// TwinCAT 3 PLC project PLC_01
// ProgramVersion: 3.1.4020.4
// libraries:
//   Tc2_Standard, * (Beckhoff Automation GmbH)
//   Tc2_System, * (Beckhoff Automation GmbH)
//   Tc2_Utilities, * (Beckhoff Automation GmbH)
//   Tc3_Module, * (Beckhoff Automation GmbH)
//   VisuDialogs, * (System)
// project tree:
//   DUTs/System/ ST_Ctrl.TcDUT, ST_Error.TcDUT, ST_Status.TcDUT
//   / GlobalTextList.TcGTLO, PlcTask.TcTTO, Visualisierungsmanager.TcVMO (not stored), VISU_TASK.TcTTO
//   GVLs/ GVL_Const.TcGVL
//   POUs/700 File/ FB_DirectoryRead.TcPOU, FB_openPDF.TcPOU
//   POUs/800 Visualisierung/ FB_TrendBuffer.TcPOU, PRG_System.TcPOU, PRG_Visualisierung.TcPOU
//   POUs/ FB_PWM.TcPOU, FUN_String_to_Time.TcPOU, MAIN.TcPOU, PRG_CAN.TcPOU
//   VISUs/ Frame_Trend_Einzel.TcVIS, Visualization.TcVIS
// real-time tasks:
//   TASK PlcTask: cycle T#10ms, priority 20, ADS port 350
//   TASK VISU_TASK: cycle T#200000us, priority 30, ADS port 351
// I/O:
//   DEVICE Gerät 1 (EtherCAT), AmsNetId 5.42.100.143.2.1
//     Klemme 1 (EK1200) [EK1200-5000 EtherCAT Netzteil (2A E-Bus)]
//       Klemme 2 (EL2008) [EL2008 8K. Dig. Ausgang 24V, 0.5A]
//       Klemme 3 (EL2008) [EL2008 8K. Dig. Ausgang 24V, 0.5A]
//       Klemme 4 (EL4104) [EL4104 4Ch. Ana. Ausgang 0-10V, 16bit]
//       Klemme 5 (EL3162) [EL3162 2K. Ana. Eingang 0-10V]
//       Klemme 6 (EL6751) [EL6751 (CANopen Master)]
//       Klemme 7 (EL9011) [EL9011 Endklemme]
//   DEVICE Gerät 2 (EL6751), AmsNetId 5.42.100.143.3.1
//     Box 8 (CANopen Node)
// variable links:
//   PLC_01/PLC_01 Instance <-> Device 1 (EtherCAT)/Term 1 (EK1200)/Term 2 (EL2008)
//     PlcTask Outputs/MAIN.ATQ_output1 <-> Channel 1/Output
//     PlcTask Outputs/MAIN.ATQ_output2 <-> Channel 2/Output
//   PLC_01/PLC_01 Instance <-> Device 1 (EtherCAT)/Term 1 (EK1200)/Term 6 (EL6751)
//     PlcTask Inputs/MAIN.ATI_input1 <-> WcState/WcState
//   PLC_01/PLC_01 Instance <-> Device 2 (EL6751)/Box 8 (CANopen Node)
//     PlcTask Inputs/PRG_CAN.CAN_master_Rx_ATI_1040 <-> TxPDO 1/Inputs/#10.40
//     PlcTask Inputs/PRG_CAN.CAN_master_Rx_ATI_201 <-> TxPDO 1/Inputs/#2.01
//     PlcTask Outputs/PRG_CAN.CAN_master_Tx_ATQ_121 <-> RxPDO 1/Outputs/#1.21
//     PlcTask Outputs/PRG_CAN.CAN_master_Tx_ATQ_642 <-> RxPDO 1/Outputs/#6.42

CONFIGURATION PLC_01
    RESOURCE PLC ON TwinCAT3
        TASK PlcTask(INTERVAL := T#10ms, PRIORITY := 20);
        TASK VISU_TASK(INTERVAL := T#200000us, PRIORITY := 30);
        PROGRAM MAIN WITH PlcTask : MAIN;
        PROGRAM VisuElems_Visu_Prg WITH VISU_TASK : VisuElems.Visu_Prg;
    END_RESOURCE
END_CONFIGURATION

// ---- DUTs/System/ST_Ctrl.TcDUT
TYPE ST_Ctrl :
STRUCT
	Init: BOOL;
	Execute: BOOL;
	Reset: BOOL;
	

END_STRUCT
END_TYPE

// ---- DUTs/System/ST_Error.TcDUT
TYPE ST_Error :
STRUCT
	Err				: BOOL;			// Hier wird das Auftreten eines Fehlers signalisiert
	ID				: UDINT;		// Hier wird eine codierte Fehlermeldung bereitgestellt - mehrere Fehler gleichzeitig möglich
	Ort				: STRING;		// Bei gesetztem Error die Angabe Ort
	OrtID			: UDINT;		// Bei gesetztem Error die Angabe Ort Id
	Modul			: STRING;		// Bei gesetztem Error die Angabe Modul
	ModulID			: UDINT;		// Bei gesetztem Error die Angabe Modul Id
	SubModul		: STRING;		// Bei gesetztem Error die Angabe SubModul
	SubModulID		: UDINT;		// Bei gesetztem Error die Angabe SubModul Id
	Text			: STRING;		// Hier wird die erste Fehlermeldung als Text bereitgestellt - nur eine Meldung möglich
	TextID			: UDINT;		// Hier wird die erste Fehlermeldung als Text bereitgestellt - nur eine Meldung möglich
	SystemTime		: STRING;		// Bei gesetztem Error die Angabe der Zeit = Systemzeit, String = YYYY-MM-DD-hh:mm:ss:xxx
													

END_STRUCT
END_TYPE

// ---- DUTs/System/ST_Status.TcDUT
TYPE ST_Status :
STRUCT
	InitOk:BOOL;
	Done:BOOL;
	Busy:BOOL;
	stError:ST_Error;

END_STRUCT
END_TYPE

// ---- GVLs/GVL_Const.TcGVL
VAR_GLOBAL CONSTANT
	
//Trend Darstellung
	gc_max_Plots				: INT:=2; 	//Maximale Anzahl an FB Trend Instanzen (und somit an möglichen Plots)
	gc_Max_ITEMS				: INT:=500; //Maximale Anzahl an Items (bei 50 wird nur das halbe Histogramm gefüllt)

//Directory read
	gcFileList_Min		: UINT:=1;						(*First line of the table*)
	gcFileList_Max		: UINT:=100;					(*Last line of the table*)
END_VAR

// ---- POUs/MAIN.TcPOU
PROGRAM MAIN
VAR

	
	//Digital I/O
	ATI_input1 AT%I* : BOOL;
	ATI_input2 AT%I* : BOOL;
	
	ATQ_output1 AT%Q* : BOOL;
	ATQ_output2 AT%Q* : BOOL;
	
	

	
	
	
	
	//zu öffnende Datei
	dateiname:STRING:='C:\Temp\B.pdf';		//Variante 1
	dateiname2:STRING:='';									//Variante 2 (wird aus Pfad und gefundener Datei zusammengesetzt
	Pfadname: STRING:='C:\Temp\';							//zu durchsuchender Pfad
	dateiindex:UINT;										//index der zu wählenden Datei
	
	//PWM Zeiten
	szeit_on:STRING:='500';		//als String (Eingabe in Visu)
	tzeit_on:TIME;				//als Zeit (umgerechnet mit der Funktion String_to_Time)
	szeit_off:STRING:='500';
	tzeit_off:TIME;
	
	// Auswahlbox
	auswahl_index: INT;			//gewählter index
	auswahl : ARRAY[0..2] OF STRING:=['Ein', 'Aus', 'PWM'];	//zur Auswahl stehende Betriebsarten
	
	//Instanzen:
	fbpwm: FB_PWM;
	
	fbdirectoryRead		: FB_DirectoryRead;
	fbopenPDF		 	: FB_openPDF;
	fbopenPDF2			: FB_openPDF;
	
	
	ctrl_pdf_1: ST_Ctrl;
	ctrl_pdf_2: ST_Ctrl;
	ctrl_readdir: ST_Ctrl;
	status:ST_Status;
	
	
	step: INT;
	change: BOOL;
	step_last: INT;
	
	plot : ARRAY[1..GVL_Const.gc_max_Plots] OF REAL;
	
	
END_VAR


PRG_System();

//Aufruf des Programms zum öffnen der PDF Datei (direkte Pfadangabe)
fbopenPDF(
	ctrl:=ctrl_pdf_1,				//ctrl.Execute startet den Öffnen Vorgang
	dateiname:=dateiname,	//Pfad zu der zu öffnenden Datei
	status=>status );		//Rückgabe des Status

//Über Verzeichnis auslesen
fbdirectoryRead(ctrl:=ctrl_readdir , PathName:=Pfadname , status=> );
//Dateiauswählen
dateiname2:=Tc2_Standard.CONCAT(Pfadname,fbdirectoryRead.List[dateiindex]);
//und öffnen
fbopenPDF2(
	ctrl:=ctrl_pdf_2,		//ctrl.Execute startet den Öffnen Vorgang
	dateiname:=dateiname2,	//Pfad zu der zu öffnenden Datei
	status=>status );		//Rückgabe des Status

//Aufruf des Plot Diagramms	
plot[1]:=BOOL_TO_REAL(ATQ_output1);
plot[2]:=BOOL_TO_REAL(ATQ_output2);
PRG_Visualisierung(plot:=plot , TaskCycleTime_ms:=PRG_System.TaskCycleTime_ms );	

//Betriebsartenauswahl
CASE step OF
	100: //idle
		IF auswahl_index<>step_last THEN
			CASE auswahl_index OF
			0:	step:=0;
				step_last:=0;
			1: 	step:=1;
				step_last:=1;
			2:  step:=2;
				step_last:=2;
			END_CASE
		END_IF
		
	0: //Ein
		ATQ_output1:=TRUE;
		ATQ_output2:=TRUE;
		step:=100;
		
	1: // Aus
		ATQ_output1:=FALSE;
		ATQ_output2:=FALSE;
		step:=100;
		
	2: //PWM	
		//UMrechnung der String in Zeiten
		tzeit_on:=FUN_String_to_Time(text:=szeit_on);
		tzeit_off:=FUN_String_to_Time(text:=szeit_off);
		
		fbpwm(
			tHightime:=tzeit_on,	//High Zeit
			tLowtime:=tzeit_off);	//Low Zeit
		ATQ_output2:=fbpwm.output;	//Schreiben des Ausgangs
		
		IF auswahl_index<>2 THEN
			step:=100;
		END_IF
END_CASE


PRG_CAN();

END_PROGRAM

// ---- POUs/FB_PWM.TcPOU
FUNCTION_BLOCK FB_PWM
VAR_INPUT
	tHightime	: TIME;
	tLowtime	: TIME;

END_VAR
VAR_OUTPUT
	output		: BOOL;
END_VAR
VAR
 	timer 		: Tc2_Standard.TON;
	step		: INT;
END_VAR


CASE step OF
	0:	//low
		output:=FALSE;
		timer(IN:=TRUE , PT:=tLowtime , Q=> , ET=> );
		IF timer.Q THEN
			timer(IN:=FALSE);
			step:=1;
		END_IF
		
	1: 	//high
		output:=True;
		timer(IN:=TRUE , PT:=tHightime , Q=> , ET=> );
		IF timer.Q THEN
			timer(IN:=FALSE);
			step:=0;
		END_IF
END_CASE

END_FUNCTION_BLOCK

// ---- POUs/700 File/FB_DirectoryRead.TcPOU
FUNCTION_BLOCK FB_DirectoryRead
VAR_INPUT
	ctrl: ST_Ctrl;
	PathName : STRING;
END_VAR
VAR_OUTPUT
	status		: ST_Status;
	List		: ARRAY[gcFileList_Min..gcFileList_Max] OF STRING;
END_VAR
VAR
	nstep: INT;
	
	fbEnumFindFileList			: FB_EnumFindFileList;
	sPathName: STRING(255);
	FindList 						: ARRAY[gcFileList_Min..gcFileList_Max] OF ST_FindFileEntry;
	nindex: UINT;
END_VAR

CASE nstep OF
0: //init
	status.InitOk:=TRUE;
	
	IF status.InitOk THEN
		nstep:=1;
	END_IF
	
1: //idle
	
	IF ctrl.Execute THEN
		status.Done:=FALSE;
		status.Busy:=TRUE;
		nstep:=2;
	END_IF
	
2: //lesen öffnen
	sPathName:=CONCAT(PathName, '*.pdf') ;	

	fbEnumFindFileList(
		sNetId:='',
		sPathName:=sPathName ,
		eCmd:=eEnumCmd_First ,
		pFindList:=ADR(FindList) ,
		cbFindList:=SIZEOF(FindList) ,
		bExecute:=TRUE ,
		tTimeout:= ,
		bBusy=> ,
		bError=> ,
		nErrID=> ,
		bEOE=>  ,
		nFindFiles=> );

	// Abfrage ob Fertig und kein Fehler
	IF NOT fbEnumFindFileList.bBUSY THEN
		status.Busy:=FALSE;
		IF NOT fbEnumFindFileList.bError THEN
			fbEnumFindFileList(bExecute:=FALSE);
			IF fbEnumFindFileList.bEOE THEN
				
				FOR nindex:=gcFileList_Min TO gcFileList_Max DO
					List[nindex]:=FindList[nindex].sFileName;
				END_FOR
				
				nstep:=3;
			END_IF
		ELSE
			nstep:=99; //Fehler
		END_IF
		
	END_IF	
	
	
3: //fertig
	status.Busy:=FALSE;
	status.Done:=TRUE;
	IF NOT ctrl.Execute THEN
		nstep:=1;
	END_IF

8: //reset
	status.stError.Err:=FALSE;
	fbEnumFindFileList(bExecute:=FALSE);
	nstep:=0;

99: //Fehler
	status.stError.Err:=TRUE;
	status.stError.ID:=fbEnumFindFileList.nErrID;
	status.Busy:=FALSE;
	
	IF ctrl.Reset THEN
		nstep:=8;
	END_IF
	
END_CASE

END_FUNCTION_BLOCK

// ---- POUs/700 File/FB_openPDF.TcPOU
FUNCTION_BLOCK FB_openPDF
VAR_INPUT
	ctrl: ST_Ctrl;
	dateiname:STRING:='C:\Temp\Beispielprojekt.pdf';
END_VAR

VAR_OUTPUT
	status: ST_Status;
END_VAR

VAR
	fbntstartprozess: NT_StartProcess;
	nstep: INT;
END_VAR

CASE nstep OF
0: //init
	status.InitOk:=TRUE;
	
	IF status.InitOk THEN
		nstep:=1;
	END_IF
	
1: //idle
	
	IF ctrl.Execute THEN
		status.Done:=FALSE;
		status.Busy:=TRUE;
		nstep:=2;
	END_IF
	
2: //PDF öffnen
	
	fbntstartprozess(
		NETID:='' , 
		(*64 Bit*)
		//PATHSTR:='C:\Program Files (x86)\Adobe\Acrobat Reader DC\Reader\AcroRd32.exe' , //Pfad des PDF Viewers
		//DIRNAME:='C:\Program Files (x86)\' , 											//Verzeichnis des Viewers
		(**)
		(*32 Bit*)
		PATHSTR:='C:\Program Files\Adobe\Acrobat Reader DC\Reader\AcroRd32.exe' , //Pfad des PDF Viewers
		DIRNAME:='C:\Program Files\' , 											//Verzeichnis des Viewers
		(**)
		COMNDLINE:=dateiname ,  												//zu öffnende Datei
		START:= TRUE, 
		TMOUT:= , 																//Default wert
		BUSY=> , 
		ERR=> , 
		ERRID=> );

	// Abfrage ob Fertig und kein Fehler
	IF NOT fbntstartprozess.BUSY THEN
		status.Busy:=FALSE;
		IF NOT fbntstartprozess.ERR THEN
			nstep:=3;
			fbntstartprozess(START:=FALSE);
		ELSE
			nstep:=99; //Fehler
		END_IF
		
	END_IF	
	
	
3: //fertig
	status.Busy:=FALSE;
	status.Done:=TRUE;
	IF NOT ctrl.Execute THEN
		nstep:=1;
	END_IF

8: //reset
	status.stError.Err:=FALSE;
	fbntstartprozess(START:=FALSE);
	nstep:=0;

99: //Fehler
	status.stError.Err:=TRUE;
	status.stError.ID:=fbntstartprozess.ERRID;
	status.Busy:=FALSE;
	
	IF ctrl.Reset THEN
		nstep:=8;
	END_IF
	
END_CASE

END_FUNCTION_BLOCK

// ---- POUs/800 Visualisierung/PRG_System.TcPOU
PROGRAM PRG_System
VAR_INPUT
	bWritePersistentData			: BOOL; //True, wenn persistente Daten geschrieben werden sollen
	bStartExplorer					: BOOL; //True, wenn Window Explorer geöffnet werden soll
	bShutdown						: BOOL; //True, wenn Rechner runtergefahren werden soll
END_VAR
VAR_OUTPUT
	SystemTime_ms					: STRING;
	TaskCycleTime_ms				: UDINT;
	SystemTime_DT					: DT;
	nCountPersistentData			: UINT;			//Zähler der persitenten Schreibvorgänge
	stError							: ST_Error;
END_VAR
VAR
	fbGetCurTaskIdx					: GETCURTASKINDEX;
	fbRegQueryValue					: FB_RegQueryValue;

	fbLocalSystemTime				: FB_LocalSystemTime;
	fbSetLocalTime 					: NT_SetLocalTime;
	fbGetTimeZoneInformation 		: FB_GetTimeZoneInformation;
	TaskCycleTime_ns				: UDINT;
	
	LastExecTime_ms					: UDINT;
	rtrigCycleTimeExceeded			: R_TRIG;
	
	
	rTrigPersistentDataWrite		: R_TRIG;
	fbWritePersistentData			: FB_WritePersistentData;
	rTrigPersistentDataDone			: F_TRIG;

	bFirstCycle						: BOOL;
	CountCycleTimeExceeded	: UINT;
	PeakHoldLastExectime_ms: UDINT;
	
	fbShutdown						: NT_Shutdown;
	fbStartProcess					: NT_StartProcess;
	
END_VAR

// ---------------------------------------------------------------------------------------------------------------------
// _AppInfo
// ---------------------------------------------------------------------------------------------------------------------
 (*
 TYPE PlcAppSystemInfo

	Each PLC provides a global instance of this type named '_AppInfo'.
	The corresponding namespace is 'TwinCAT_SystemInfoVarList'. For example this has to be added inside a library.

--------------------------------------------------------------------------------------------------------------------------------------------------------------------------------------------------------------------------------------------------
TYPE PlcAppSystemInfo
STRUCT
         ObjId             		: OTCID;				// 	object ID of the PLC project instance
         TaskCnt           		: UDINT;				// The number of tasks in the actual runtime system.
         OnlineChangeCnt   		: UDINT;				// The number of online changes made since the last complete download.
         Flags             		: DWORD;				// Reserved for future use
         AdsPort           		: UINT;					// ADS port of PLC application
         BootDataLoaded    		: BOOL;					// PERSISTENT variables: LOADED (without error)
         OldBootData       		: BOOL;					// PERSISTENT variables: INVALID (the back-up copy was loaded, since no valid data was present)
         AppTimestamp      		: DT;					// Date and time of application start
         KeepOutputsOnBP   		: BOOL;					// The flag can be set to avoid that the outputs are zero-filled if a breakpoint is reached. The task keeps running. Only the execution of PLC code is interrupted.
         TComSrvPtr        		: ITComObjectServer;	// Pointer to TcCOM Object Server
         AppName           		: STRING(63);			// TwinCAT generated name containing the port number
         ProjectName       		: STRING(63);			// The name of the PLC project.
END_STRUCT
END_TYPE
 
If the variable runTimeNo was used under TwinCAT 2, the program code has to be changed.
Sample:
Usage under TwinCAT 2:   nPlcAdsPort := 801 + (SystemInfo.runTimeNo - 1) * 10;
Usage under TwinCAT 3:   nPlcAdsPort := _AppInfo.AdsPort;
 *)
 
 _AppInfo.ObjId:=_AppInfo.ObjId;
 _AppInfo.TaskCnt:=_AppInfo.TaskCnt;
 _AppInfo.OnlineChangeCnt:=_AppInfo.OnlineChangeCnt;
 _AppInfo.Flags:=_AppInfo.Flags;
 _AppInfo.AdsPort:=_AppInfo.AdsPort;
 _AppInfo.BootDataLoaded:=_AppInfo.BootDataLoaded;
 _AppInfo.OldBootData:=_AppInfo.OldBootData;
 _AppInfo.AppTimestamp:=_AppInfo.AppTimestamp;
 _AppInfo.KeepOutputsOnBP:=_AppInfo.KeepOutputsOnBP;
 _AppInfo.TComSrvPtr:=_AppInfo.TComSrvPtr;
 _AppInfo.AppName:=_AppInfo.AppName;
 _AppInfo.ProjectName:=_AppInfo.ProjectName;


// ---------------------------------------------------------------------------------------------------------------------
// _TaskInfo
// ---------------------------------------------------------------------------------------------------------------------
 (*
 TYPE PlcTaskSystemInfo

	Each PLC provides an array of global instances of this type named '_TaskInfo[]'.
	The corresponding namespace is 'TwinCAT_SystemInfoVarList'. For example this has to be added inside a library.

--------------------------------------------------------------------------------------------------------------------------------------------------------------------------------------------------------------------------------------------------
{attribute 'Namespace' := 'PLC'}
TYPE PlcTaskSystemInfo
STRUCT
         ObjId             		: OTCID;				// 	Object ID of task reference calling the PLC program.
         CycleTime         		: UDINT;				// Cycletime set in the task configuration in parts of 100ns.
         Priority          		: UINT;					// Priority set in the task configuration.
         AdsPort           		: UINT;					// 	ADS port of Task
         CycleCount        		: UDINT;				// Cyclecounter.
         DcTaskTime        		: LINT;					// Distributed Clock System Time. It remains constant for a task duration.
         LastExecTime      		: UDINT;				// Needed cycletime for the last cycle in parts of 100ns.
         FirstCycle        		: BOOL;					// The variable is TRUE in the first cycle of the task.
         CycleTimeExceeded 		: BOOL;					// 	The variable is TRUE if the runtime of the task exceeds the cycletime set in task configuration.
         TaskName          		: STRING(63);			// Contains the name of the task
END_STRUCT
END_TYPE

Sample:
fbGetCurTaskIdx();                                                                           // declared as: fbGetCurTaskIdx : GETCURTASKINDEX;
nCycleTime := _TaskInfo[fbGetCurTaskIdx.index].CycleTime;
*)
 
 fbGetCurTaskIdx();                                                                           // declared as: fbGetCurTaskIdx : GETCURTASKINDEX;

 _TaskInfo[fbGetCurTaskIdx.index].ObjId:=_TaskInfo[fbGetCurTaskIdx.index].ObjId;
 _TaskInfo[fbGetCurTaskIdx.index].CycleTime:=_TaskInfo[fbGetCurTaskIdx.index].CycleTime;
 _TaskInfo[fbGetCurTaskIdx.index].Priority:=_TaskInfo[fbGetCurTaskIdx.index].Priority;
 _TaskInfo[fbGetCurTaskIdx.index].AdsPort:=_TaskInfo[fbGetCurTaskIdx.index].AdsPort;
 _TaskInfo[fbGetCurTaskIdx.index].CycleCount:=_TaskInfo[fbGetCurTaskIdx.index].CycleCount;
 _TaskInfo[fbGetCurTaskIdx.index].DcTaskTime:=_TaskInfo[fbGetCurTaskIdx.index].DcTaskTime;
 _TaskInfo[fbGetCurTaskIdx.index].LastExecTime:=_TaskInfo[fbGetCurTaskIdx.index].LastExecTime;
 _TaskInfo[fbGetCurTaskIdx.index].FirstCycle:=_TaskInfo[fbGetCurTaskIdx.index].FirstCycle;
 _TaskInfo[fbGetCurTaskIdx.index].CycleTimeExceeded:=_TaskInfo[fbGetCurTaskIdx.index].CycleTimeExceeded;
 _TaskInfo[fbGetCurTaskIdx.index].TaskName:=_TaskInfo[fbGetCurTaskIdx.index].TaskName;
 
// ---------------------------------------------------------------------------------------------------------------------
// Zykluszeit mit Spitzenwert 8Peak Hold)
// ---------------------------------------------------------------------------------------------------------------------
TaskCycleTime_ns:=_TaskInfo[fbGetCurTaskIdx.index].CycleTime/10;
TaskCycleTime_ms:=_TaskInfo[fbGetCurTaskIdx.index].CycleTime/10000;
LastExecTime_ms:=_TaskInfo[fbGetCurTaskIdx.index].LastExecTime/10000;
IF PeakHoldLastExectime_ms<LastExecTime_ms THEN
	PeakHoldLastExectime_ms:=LastExecTime_ms;
END_IF

// ---------------------------------------------------------------------------------------------------------------------
// Zykluszeitüberschreitungen zählen
// ---------------------------------------------------------------------------------------------------------------------
rtrigCycleTimeExceeded(CLK:=_TaskInfo[fbGetCurTaskIdx.index].CycleTimeExceeded , Q=> );
IF rtrigCycleTimeExceeded.Q THEN
	CountCycleTimeExceeded:=CountCycleTimeExceeded+1;
END_IF

// ---------------------------------------------------------------------------------------------------------------------
// PLC First Cycle
// ---------------------------------------------------------------------------------------------------------------------
bFirstCycle:=_TaskInfo[fbGetCurTaskIdx.index].FirstCycle;

// ---------------------------------------------------------------------------------------------------------------------
// Windows Systemzeit 
// ---------------------------------------------------------------------------------------------------------------------
 fbLocalSystemTime(
	sNetID:='' ,
	bEnable:=TRUE ,
	dwCycle:= ,
	dwOpt:= ,
	tTimeout:=DEFAULT_ADS_TIMEOUT ,
	bValid=> ,
	systemTime=> ,
	tzID=> );
IF fbLocalSystemTime.bValid THEN
	SystemTime_ms:=LEFT(SYSTEMTIME_TO_STRING(fbLocalSystemTime.systemTime),16);
	SystemTime_DT:=SYSTEMTIME_TO_DT(fbLocalSystemTime.systemTime);
END_IF

// ---------------------------------------------------------------------------------------------------------------------
// Persisten Data
// ---------------------------------------------------------------------------------------------------------------------
rTrigPersistentDataWrite(CLK:=bWritePersistentData , Q=> );
fbWritePersistentData(
	NETID:= '', 
	PORT:= _TaskInfo[fbGetCurTaskIdx.index].AdsPort , 
	START:= rTrigPersistentDataWrite.Q , 
	TMOUT:= DEFAULT_ADS_TIMEOUT , 
	MODE:= SPDM_2PASS, 
	BUSY=> , 
	ERR=> , 
	ERRID=> );
rTrigPersistentDataDone(CLK:=fbWritePersistentData.BUSY , Q=> );
IF rTrigPersistentDataDone.Q THEN
	nCountPersistentData:=nCountPersistentData+1;
END_IF

// ---------------------------------------------------------------------------------------------------------------------
// Windows / Explorer
// ---------------------------------------------------------------------------------------------------------------------
fbStartProcess(
	NETID:='' , 
	PATHSTR:='C:\Windows\Explorer.exe' , 
	DIRNAME:= , 
	COMNDLINE:= , 
	START:=bStartExplorer , 
	TMOUT:=DEFAULT_ADS_TIMEOUT , 
	BUSY=> , 
	ERR=> , 
	ERRID=> );





// ---------------------------------------------------------------------------------------------------------------------
// Windows / PC ausschalten
// ---------------------------------------------------------------------------------------------------------------------
fbShutdown(
	NETID:='' , 
	DELAY:=5 , 
	START:=bShutdown , 
	TMOUT:=DEFAULT_ADS_TIMEOUT , 
	BUSY=> , 
	ERR=> , 
	ERRID=> );


// ---------------------------------------------------------------------------------------------------------------------
// ENDE
// ---------------------------------------------------------------------------------------------------------------------

METHOD GetSystemTime : DT
VAR_INPUT
END_VAR
GetSystemTime:=SystemTime_DT;
END_METHOD

END_PROGRAM

// ---- POUs/800 Visualisierung/PRG_Visualisierung.TcPOU
PROGRAM PRG_Visualisierung
VAR_INPUT
	plot : ARRAY[1..GVL_Const.gc_max_Plots] OF REAL; 	//Array von den Werten (in REAL) die geplottet werden sollen
	TaskCycleTime_ms : UDINT;							//Zykluszeit in ms ( z.B. aus PRG_System)
END_VAR
VAR_OUTPUT
END_VAR
VAR
	
	fbpwmTrend :ARRAY[1..GVL_Const.gc_max_Plots] OF  FB_TrendBuffer;
	
	nindex:INT;
	
END_VAR


//Aufruf des FB zur Erzeugung des Trends
FOR nindex:=1  TO GVL_Const.gc_max_Plots DO  
	
	fbpwmTrend[nindex](
		uiValue:= plot[nindex],  						// Eingangssignal
		dtSystemTime:= PRG_System.GetSystemTime(), 
		tCycleTime:= UDINT_TO_TIME(TaskCycleTime_ms), 	// Zykluszeit
		bReverseFilll:= , 
		count=> , 
		dtFirstTimeStamp=> , 
		dtLastTimeStamp=> 
	);
END_FOR

END_PROGRAM

// ---- POUs/800 Visualisierung/FB_TrendBuffer.TcPOU
FUNCTION_BLOCK FB_TrendBuffer
VAR_INPUT
	uiValue 		: REAL;			//Zu plottender Wert
	dtSystemTime 	: DT;
	tCycleTime 		: TIME;			//Zyklus Zeit
	bReverseFilll 	: BOOL;			//False: von rechts nach links , True von Links nach rechts verschieben
END_VAR
VAR_OUTPUT
	count 		     : UINT;
	dtFirstTimeStamp : DT;
	dtLastTimeStamp  : DT;
END_VAR

VAR
	itemValue 		 : ARRAY[1..GVL_Const.gc_Max_ITEMS] OF REAL; 		//Array was an das Histogramm weitergegeben werden muss
	itemTimeStamp    : ARRAY[1..GVL_Const.gc_Max_ITEMS] OF DT;

	cycle 			 : TOF;
	bFullBuffer 	 : BOOL;
END_VAR

(*
- Pro zu Plottendem Wert ist eine Instanz anzulegen
- uiValue ist die Eingangsvariable
- itemValue ist das zu plottende Array

*)



IF NOT cycle.Q THEN
	count := MIN(count +1,GVL_Const.gc_Max_ITEMS);
	CASE BOOL_TO_INT(bReverseFilll) OF
	0:
		IF bFullBuffer THEN
			MEMCPY(ADR(itemValue),ADR(itemValue)+SIZEOF(itemValue[GVL_Const.gc_Max_ITEMS]),SIZEOF(itemValue)-SIZEOF(itemValue[GVL_Const.gc_Max_ITEMS]));
			MEMCPY(ADR(itemTimeStamp),ADR(itemTimeStamp)+SIZEOF(itemTimeStamp[GVL_Const.gc_Max_ITEMS]),SIZEOF(itemTimeStamp)-SIZEOF(itemTimeStamp[GVL_Const.gc_Max_ITEMS]));
		END_IF
		bFullBuffer := (count >= GVL_Const.gc_Max_ITEMS);
		itemValue[count] := uiValue;
		itemTimeStamp[count] := dtSystemTime;
	ELSE
		MEMCPY(ADR(itemValue)+SIZEOF(itemValue[GVL_Const.gc_Max_ITEMS]),ADR(itemValue),SIZEOF(itemValue)-SIZEOF(itemValue[GVL_Const.gc_Max_ITEMS]));
		MEMCPY(ADR(itemTimeStamp)+SIZEOF(itemTimeStamp[GVL_Const.gc_Max_ITEMS]),ADR(itemTimeStamp),SIZEOF(itemTimeStamp)-SIZEOF(itemTimeStamp[GVL_Const.gc_Max_ITEMS]));
		itemValue[1] := uiValue;
		itemTimeStamp[1] := dtSystemTime;
	END_CASE
	
	dtFirstTimeStamp := itemTimeStamp[1];
	dtLastTimeStamp := itemTimeStamp[count];
END_IF

cycle(IN:=NOT cycle.Q, PT:=tCycleTime);

END_FUNCTION_BLOCK

// ---- POUs/FUN_String_to_Time.TcPOU
FUNCTION FUN_String_to_Time : Time
VAR_INPUT
	text:STRING;
END_VAR
VAR
	temp :string;
END_VAR

//zusammensetzten des Strings
temp:=Tc2_Standard.CONCAT(STR1:=Tc2_Standard.CONCAT(STR1:='T#',STR2:=text),STR2:='ms');

//Konvertierung in Zeit
FUN_String_to_Time:=STRING_TO_TIME(temp);

END_FUNCTION

// ---- POUs/PRG_CAN.TcPOU
PROGRAM PRG_CAN
VAR_INPUT

END_VAR

VAR_OUTPUT

END_VAR

VAR
//CAN test
	//wird vom Master empfangen
	CAN_master_Rx_ATI_1040 	AT%I* :DINT;	// status word
	CAN_master_Rx_ATI_201   AT%I* :DINT;	// post-ramp speed	
	
	//wird vom Master gesendet
	CAN_master_Tx_ATQ_642 	AT%Q* :DINT;	// control word
	CAN_master_Tx_ATQ_121 	AT%Q* :DINT;	// digital speed	
	

(*
	Polled channel 			Data word 	Mapping parameter 	Size(bits) 		Default mapping status
	IN  channel 0 RxPDO 	Word 0, 1 	Pr MM.10 			32 				1040 (Pr 10.40, status word)
	IN  channel 1 RxPDO 	Word 2, 3 	Pr MM.11 			32 				 201 (Pr 2.01, post-ramp speed ref)
	
	OUT channel 0 TxPDO 	Word 0, 1 	Pr MM.20 			32 				 642 (Pr 6.42, control word)
	OUT channel 1 TxPDO 	Word 2, 3 	Pr MM.21 			32 				 121 (Pr 1.21, digital speed ref 1)

*)



//Table 9.2 Control WORD BIT functions
	(*
	0 ENABLE Set to 1 to enable the drive. Resetting to 0 will immediately disable the drive,
	and the motor will coast to a stop. The external HARDWARE ENABLE signal
	must also be present before the drive can be enabled.
	*)
	benable:BOOL;
	(*
	1 RUN FWD Set to 1 (with ENABLE set to 1) to run the motor in the forward direction. When
	reset to 0, the drive will decelerate the motor to a controlled stop.
	*)
	brunFWD:BOOL;
	(*
	2* JOG FWD
	Set to 1 to jog the motor forward. This signal needs to be used in conjunction
	with the ENABLE bit. This signal is overridden by a RUN, RUN REV or RUN
	FWD signal.
	*)
	bJogFWD:BOOL;
	(*	
	3 RUN REVSet to 1 (with ENABLE set to 1) to run the motor in the reverse direction. When
	reset to 0, the drive will decelerate the motor to a controlled stop.
	*)
	bRunREV:BOOL;
	(*
	4 FWD REV Set to 1 to select the reverse direction. Set to 0 to run in the forward direction.
	The RUN signal is used to start and stop the motor.
	*)
	bFwdREV:BOOL;
	(*
	5 RUN
	Set to 1 to run the motor. FWD REV is used to select the direction of motor
	rotation. When reset to 0, the drive will decelerate the motor to a controlled
	stop.
	*)
	bRun:BOOL;
	(*
	6* NOT	STOP
	Set to 1 to allow the sequencing bit in the drive to be latched. Refer to the drive
	Advanced User Guide for more details. If NOT STOP is zero, all latches are
	cleared and held at 0. Pr 6.04 must be correctly set for this to function.
	*)
	bNotStop:BOOL;
	(*
	7 AUTOSet to 1 to enable fieldbus control of the drive Control Word. The Control Word
	Enable (Pr 6.43) must also be set to 1. When reset to 0, the drive will operate
	under terminal control.
	*)
	bAutoSet:BOOL;
	(*
	8 REMOTE
	Set to 1 to select digital speed reference 1 (Pr 1.21), and to 0 to select analog
	reference 1 (Pr 1.36). REMOTE directly controls Pr 1.42, so reference selector
	(Pr 1.14) and preset selector (Pr 1.15) must both be set to 0 (default) for the
	REMOTE bit to work properly.
	*)
	bRemote:BOOL;
	(*
	9* JOG REV
	Set to 1 to jog the motor in reverse. This signal needs to be used in conjunction
	with the ENABLE bit. This signal is overridden by a RUN/RUN REV/RUN FWD
	command.
	*)
	bJogREV:BOOL;
	(*
	10 Reserved -
	11 Reserved -
	*)
	
	(*
	12 TRIP
	Set to 1 to trip the drive at any time. The trip display on drive will be “CL.bit”
	and the trip code will be 35. AUTO (b7) has no effect on this function. The trip
	cannot be cleared until TRIP is reset to 0.
	*)
	bTrip:BOOL;
	(*
	13 RESET
	A 0-1 transition of the RESET bit will reset the drive from a trip condition. If the
	reason for the trip is still present, or another fault condition has been detected,
	the drive will immediately trip again. When resetting the drive, it is
	recommended to check the status word to ensure that the reset was
	successful, before attempting to re-start the drive.
	*)
	bReset:BOOL;
	(*
	14* KEYPAD	WDOG
	This watchdog is provided for an external keypad or other devices where a
	break in the communication link must be detected. The watchdog system can
	be enabled and/or serviced if this bit is changed from zero to one while the
	control word enabled.
	Once the watchdog is enabled it must be serviced at least once every second
	or an “SCL” trip will occur. The watchdog is disabled when an “SLC” trip
	occurs, and so it must be re-enabled when the trip is reset. 
	*)
	bKeypadWDOG:BOOL;
	
//Table 9.3 Drive status word bit functions
	(*
	0 Drive ok Pr 10.01 Indicates the drive is not in the trip state.
	*)
	bDriveOK:BOOL;
	(*
	1 Drive active Pr 10.02 Indicates that the output stage of the drive is active.
	*)
	bDriveActive:BOOL;
	(*
	2 Zero speed Pr 10.03
	In Open Loop mode, zero speed indicates that the
	absolute value of the post-ramp speed reference is at or
	below the zero speed threshold.
	In Closed Loop and Servo modes, zero speed indicates
	that the absolute value of speed feedback is at or below
	the zero speed threshold.
	*)
	(*
	3	Running at or	below minimum	speed	Pr 10.04
	In bipolar mode (Pr 1.10 = 1) Pr 10.04 is the same as zero
	speed, Pr 10.03 (see above).
	In unipolar mode, Pr 10.04 is set if the absolute value of
	the post-ramp speed reference (Pr 2.01) or speed
	feedback (Pr 3.02) is at or below minimum speed + 0.5Hz
	or 5rpm (minimum speed is defined by Pr 1.07). This
	parameter is only set if the drive is running.
	*)
	(*
	4 Below set	speed Pr 10.05
	Only set if the drive is running at below set speed. Refer
	to Pr 3.06, Pr 3.07 and Pr 3.09 in the drive User Guide for
	more details.
	*)
	(*
	5 At speed Pr 10.06 Only set if the drive is running at set speed. Refer to
	Pr 3.06, Pr 3.07 and Pr 3.09 in the drive User Guide.
	*)
	(*
	6 Above set
	speed Pr 10.07
	Only set if the drive is running at above set speed. Refer
	to Pr 3.06, Pr 3.07 and Pr 3.09 in the drive User Guide for
	more details.
	*)
	(*
	7 Load reached Pr 10.08
	Indicates that the modulus of the active current is greater
	or equal to the rated active current, as defined in menu 4.
	Refer to the drive Advanced User Guide for more details.
	*)
	(*
	8 In current limit Pr 10.09 Indicates that the current limits are active.
	*)
	(*
	9 Regenerating Pr 10.10
	Regenerating indicates that power is being transferred
	from the motor to the drive.
	In regen mode, regenerating indicates that power is being
	transferred from the Unidrive SP to the supply.
	*)
	(*
	10 Dynamic brake
	active Pr 10.11
	Indicates that the braking IGBT is active. If the IGBT
	becomes active, this parameter will remain on for at least
	one second.
	*)
	(*
	11 Dynamic brake
	alarm Pr 10.12
	Dynamic brake alarm is set when the braking IGBT is
	active, and the braking energy accumulator is greater
	than 75%.
	*)
	(*
	12 Direction
	commanded Pr 10.13
	Direction commanded is set to 1 if the Pre-ramp speed
	reference (Pr 1.03) is negative and reset to 0 if the
	Pre-ramp speed reference is zero or positive.
	*)
	(*
	13 Direction
	running Pr 10.14
	A 0 indicates forward direction and a 1 indicates reverse
	direction. The source of this bit is Pr 2.01 for open loop
	mode and Pr 3.02 for closed loop and servo modes.
	*)
	(*
	14 Mains loss Pr 10.15
	Mains loss indicates that the drive has detected a mains
	loss from the level of the DC bus voltage. This parameter
	can only become active if mains loss ride through or
	mains loss stop modes are selected. Refer to Pr 6.03 in
	the drive Advanced User Guide for more details.
	In regen mode, mains loss is the inverse of Pr 3.07.
	*)
	(*
	15 Not Used Reserved.
*)
	
	

END_VAR


//Control word
CAN_master_Tx_ATQ_642.0:=benable; //Enable
CAN_master_Tx_ATQ_642.1:=brunFWD; 
CAN_master_Tx_ATQ_642.2:=bJogFWD; //
CAN_master_Tx_ATQ_642.3:=bRunREV; //
CAN_master_Tx_ATQ_642.4:=bFwdREV; //
CAN_master_Tx_ATQ_642.5:=bRun; //
CAN_master_Tx_ATQ_642.6:=bNotStop; //
CAN_master_Tx_ATQ_642.7:=bAutoSet; //
CAN_master_Tx_ATQ_642.8:=bRemote; //
CAN_master_Tx_ATQ_642.9:=bJogREV; //
CAN_master_Tx_ATQ_642.10:=FALSE; //
CAN_master_Tx_ATQ_642.11:=FALSE; //
CAN_master_Tx_ATQ_642.12:=bTrip; //
CAN_master_Tx_ATQ_642.13:=bReset; //
CAN_master_Tx_ATQ_642.14:=bKeypadWDOG; //
CAN_master_Tx_ATQ_642.15:=FALSE; //

//Status Word
bDriveOK:=CAN_master_Rx_ATI_1040.0;
bDriveActive:=CAN_master_Rx_ATI_1040.1;

END_PROGRAM

// ---- GlobalTextList.TcGTLO
TEXTLIST GlobalTextList
  15 = ''
  16 = '%.2f'
  5 = '%s'
  10 = 'Ausgang 1' | EN: 'Output 1'
  11 = 'Ausgang 2' | EN: 'Output 2'
  1 = 'CAN' | EN: 'CAN'
  7 = 'Deutsch' | EN: 'German'
  0 = 'Digital IO'
  8 = 'Eingang 1' | EN: 'Input 1'
  9 = 'Eingang 2' | EN: 'Input 2'
  6 = 'Englisch' | EN: 'english'
  14 = 'ms'
  4 = 'PDF'
  3 = 'PDF öffnen' | EN: 'PDF open'
  2 = 'Sprache' | EN: 'Language'
  17 = 'Verzeichnis lesen'
  12 = 'Zeit aus '
  13 = 'Zeit ein'
END_TEXTLIST

// ---- VISUs/Frame_Trend_Einzel.TcVIS
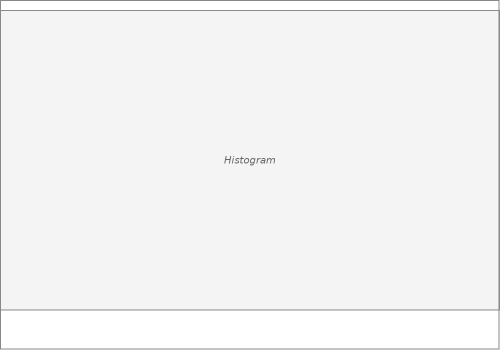
VISUALIZATION Frame_Trend_Einzel  // 500x350
VAR_IN_OUT
	itemValue : ARRAY[1..GVL_Const.gc_Max_ITEMS] OF REAL;
END_VAR
    Histogram (0,10 500x300), scale format: %.2f, scale -0.25..1.25
        p1518820177: itemValue
        p102497268: itemValue
        p788070771: ARRAY [1..GVL_Const.gc_Max_ITEMS] OF REAL
END_VISUALIZATION

// ---- VISUs/Visualization.TcVIS
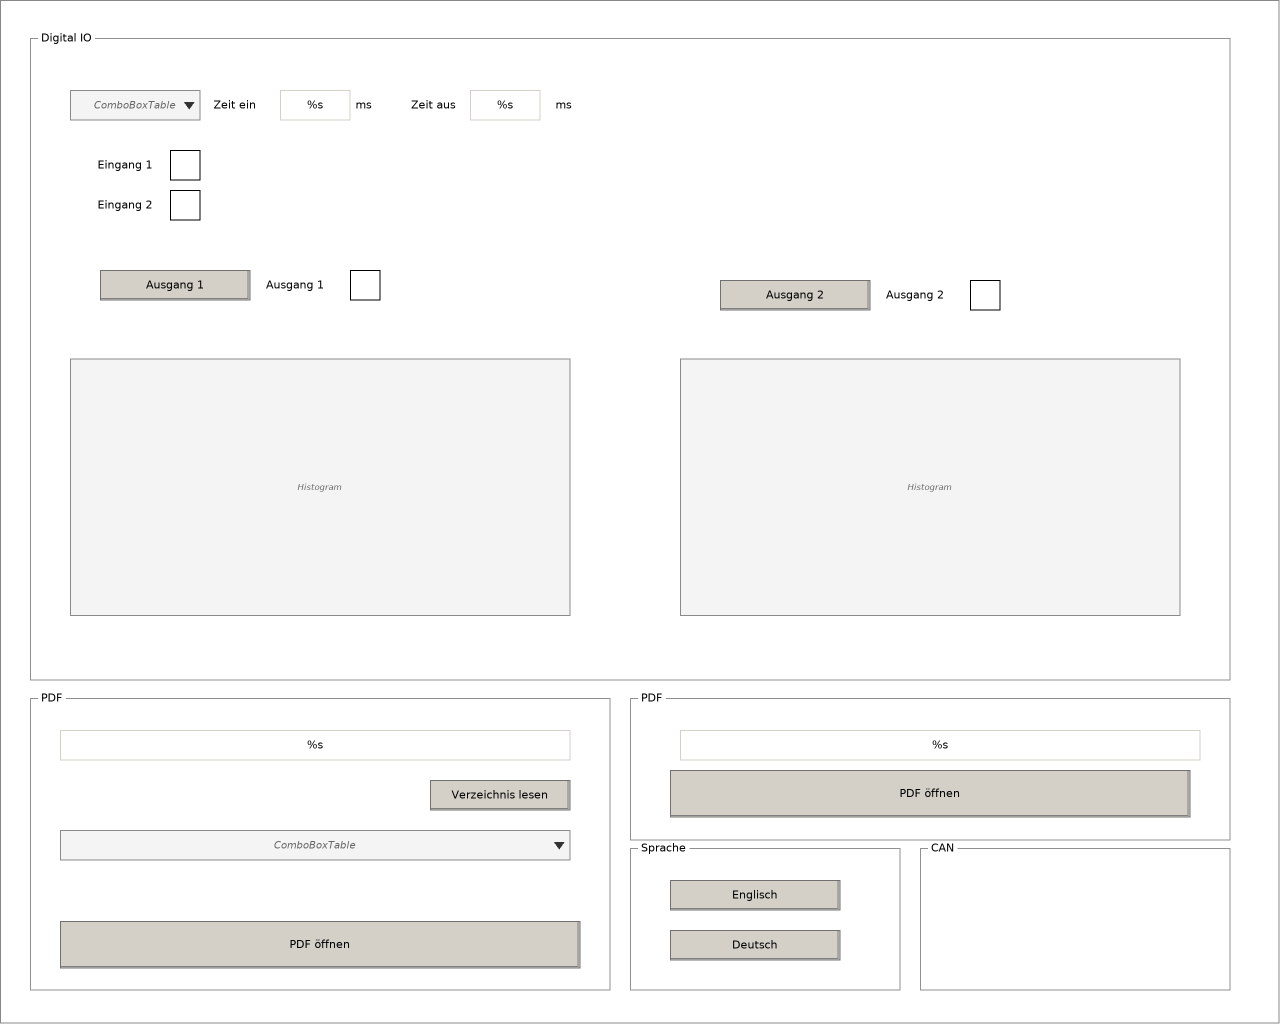
VISUALIZATION Visualization  // 1280x1024
    GroupBox (30,30 1200x650), "Digital IO"
        Rectangle (320,240 30x30), colour toggle: MAIN.ATQ_output1
        Rectangle (140,120 30x30), colour toggle: MAIN.ATI_input1
        Rectangle (140,160 30x30), colour toggle: MAIN.ATI_input2
        Rectangle (940,250 30x30), colour toggle: MAIN.ATQ_output2
        Label (40,120 110x30), "Eingang 1"
        Label (160,60 90x30), "Zeit ein"
        Label (830,250 110x30), "Ausgang 2"
        Label (210,240 110x30), "Ausgang 1"
        Button (690,250 150x30), "Ausgang 2"
            toggle MAIN.ATQ_output2
        Button (70,240 150x30), "Ausgang 1"
            toggle MAIN.ATQ_output1
        Textfield (440,60 70x30), "%s", text variable: MAIN.szeit_off
            OnMouseClick: write the text variable via Default
        Textfield (250,60 70x30), "%s", text variable: MAIN.szeit_on
            OnMouseClick: write the text variable via Default
        Label (40,160 110x30), "Eingang 2"
        Label (360,60 90x30), "Zeit aus"
        Label (320,60 27x30), "ms"
        ComboBoxTable (40,60 130x30), variable: Main.auswahl_index, data array: MAIN.auswahl
            p3854506369: MAIN.auswahl[INDEX]
        Label (520,60 27x30), "ms"
        Frame (650,320 500x300)
            shows Frame_Trend_Einzel(itemValue := PRG_Visualisierung.fbpwmTrend[2].itemValue)
        Frame (40,320 500x300)
            shows Frame_Trend_Einzel(itemValue := PRG_Visualisierung.fbpwmTrend[1].itemValue)
    GroupBox (920,840 310x150), "CAN"
    GroupBox (630,840 270x150), "Sprache"
        Button (40,40 170x30), "Englisch"
            OnMouseClick: ChangeLanguage ChangeLanguage=EN
        Button (40,90 170x30), "Deutsch"
            OnMouseClick: ChangeLanguage ChangeLanguage=DE
    GroupBox (30,690 580x300), "PDF"
        Button (400,90 140x30), "Verzeichnis lesen"
            tap MAIN.ctrl_readdir.Execute
        Textfield (30,40 510x30), "%s", text variable: MAIN.Pfadname
            OnMouseClick: write the text variable via Default
        ComboBoxTable (30,140 510x30), variable: MAIN.dateiindex, data array: MAIN.fbdirectoryRead.List
            p1892666644: MAIN.fbdirectoryRead.fbEnumFindFileList.sPathName
            p338671338: MAIN.fbdirectoryRead.fbEnumFindFileList.eCmd
            p2170511999: MAIN.fbdirectoryRead.fbEnumFindFileList.pFindList^
            p3723444502: MAIN.fbdirectoryRead.fbEnumFindFileList.cbFindList
            p1218418051: MAIN.fbdirectoryRead.fbEnumFindFileList.bExecute
            p746581629: MAIN.fbdirectoryRead.fbEnumFindFileList.tTimeout
            p3104783080: MAIN.fbdirectoryRead.fbEnumFindFileList.bBusy
            p2501879983: MAIN.fbdirectoryRead.fbEnumFindFileList.bError
            p7306298: MAIN.fbdirectoryRead.fbEnumFindFileList.nErrID
            p1933151965: MAIN.fbdirectoryRead.fbEnumFindFileList.bEOE
            p3863566920: MAIN.fbdirectoryRead.fbEnumFindFileList.nFindFiles
            p2192122294: MAIN.fbdirectoryRead.fbEnumFindFileList.fbEnum
            p400160035: MAIN.fbdirectoryRead.fbEnumFindFileList.fbTrigger
            p1265227338: MAIN.fbdirectoryRead.fbEnumFindFileList.state
            p3726181087: MAIN.fbdirectoryRead.fbEnumFindFileList.cbEntry
            p3136911649: MAIN.fbdirectoryRead.fbEnumFindFileList.nEntries
            p797552052: MAIN.fbdirectoryRead.fbEnumFindFileList.pEntry^
            p3854506369: MAIN.fbdirectoryRead.List[INDEX]
        Button (30,231 520x47), "PDF öffnen"
            tap MAIN.ctrl_pdf_2.Execute
    GroupBox (630,690 600x150), "PDF"
        Button (40,80 520x47), "PDF öffnen"
            tap MAIN.ctrl_pdf_1.Execute
        Textfield (50,40 520x30), "%s", text variable: MAIN.dateiname
            OnMouseClick: write the text variable via Default
END_VISUALIZATION
